// TIA Portal V17 export
// export: Created 2023-03-06T02:05:27.5489032Z, ExportSetting WithDefaults, DisplayName Totally Integrated Automation Portal, DisplayVersion V17 Update 4, DisplayName TIA Portal Openness, DisplayVersion V17 Update 4, DisplayName TIA Portal Version Control Interface, DisplayVersion V17, DisplayName STEP 7 Professional, DisplayVersion V17 Update 4, DisplayName STEP 7 Safety, DisplayVersion V17, DisplayName WinCC Professional, DisplayVersion V17 Update 4
TYPE "BB"
// stored: IsFailsafeCompliant false
   STRUCT
      iAssetSt : Int;
      rVcellAvg : Real;
      iTcellAvg : Int;
      iNBRConn : Int;
      rIdc : Real;
      rVcellMax : Real;
      iTcellMax : Int;
      rVcellMin : Real;
      iTcellMin : Int;
      rPdc : Real;
      rSOC : Real;
      rSOH : Real;
      rVdc : Real;
   END_STRUCT;
END_TYPE
